(* IEC 61131-3 sources: ArfBotOS/Codesys-4/ArfBotOS.fbsdev/Application.iecapp^/FUN/digital/FB_DigitalOutput.fb.st^/public, 3 files *)

(* ---- Off.meth.st ---- *)
METHOD PUBLIC Off : BOOL
VAR_INPUT
END_VAR

_Output := FALSE;
END_METHOD

(* ---- On.meth.st ---- *)
METHOD PUBLIC On : BOOL
VAR_INPUT
END_VAR

_Output := TRUE;
END_METHOD

(* ---- Toggle.meth.st ---- *)
METHOD PUBLIC Toggle : BOOL
VAR_INPUT
END_VAR

_Output := NOT _Output;
END_METHOD
